/// This function block is a container for equipment that is used by this unit.
/// Equipment is grouped by its kind (actuator, axes, io, ...).
/// It extends from [ManagedObjectContainer](xref:ZCore.ManagedObjectContainer) such that the parent
/// (= the unit itself) can be passed to equipment instances.
FUNCTION_BLOCK ScriblyEquipment EXTENDS ScriblyContainer
VAR_INPUT
  Io : ScriblyIo(_parent);
  Actuator : ScriblyActuator(_parent);
  Axis : ScriblyAxis(_parent);
  Fieldbus : ScriblyFieldbus(_parent);
  Unit : ScriblyLinkedUnit(_parent);
END_VAR

END_FUNCTION_BLOCK

(* stored: Version 1.1.0.1
   POU ScriblyEquipment: Id {dda9199d-3b7f-4fd0-8bd1-38b9dc557fbe}, SpecialFunc None *)
